// TIA Portal V18 export
FUNCTION_BLOCK "Conveyor"   // FB2, FBD
{ S7_Optimized_Access := 'TRUE' }
AUTHOR : dda
VERSION : 0.1
// stored: AutoNumber true, IsIECCheckEnabled true, IsRetainMemResEnabled false, MemoryReserve 100, SetENOAutomatically true, UDAEnableTagReadback false
   VAR_INPUT
      automaticMode { ExternalAccessible := 'False'; ExternalVisible := 'False'; ExternalWritable := 'False'} : Bool;
      manualMode { ExternalAccessible := 'False'; ExternalVisible := 'False'; ExternalWritable := 'False'} : Bool;
      jogRight { ExternalAccessible := 'False'; ExternalVisible := 'False'; ExternalWritable := 'False'} : Bool;
      run { ExternalAccessible := 'False'; ExternalVisible := 'False'; ExternalWritable := 'False'} : Bool;
   END_VAR
   VAR_OUTPUT
      conveyorRight { ExternalAccessible := 'False'; ExternalVisible := 'False'; ExternalWritable := 'False'} : Bool;
      conveyorLeft { ExternalAccessible := 'False'; ExternalVisible := 'False'; ExternalWritable := 'False'} : Bool;
   END_VAR
   VAR
      statRequest { ExternalAccessible := 'False'; ExternalVisible := 'False'; ExternalWritable := 'False'} : Bool;
      statRelease { ExternalAccessible := 'False'; ExternalVisible := 'False'; ExternalWritable := 'False'} : Bool;
   END_VAR
BEGIN

REGION Network 1 (SCL)
   // functionality: conveyor
   //
END_REGION

REGION Network 2
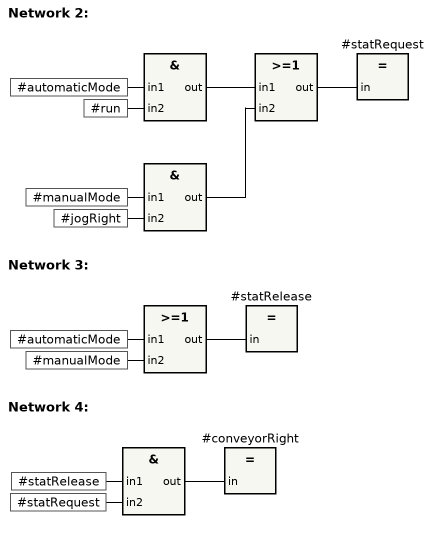
   #statRequest := (#automaticMode AND #run) OR (#manualMode AND #jogRight);
END_REGION

REGION Network 3
   #statRelease := #automaticMode OR #manualMode;
END_REGION

REGION Network 4
   #conveyorRight := #statRelease AND #statRequest;
END_REGION
END_FUNCTION_BLOCK
